PROGRAM MAIN
VAR
	tpImAPLC : TP;
END_VAR

////////////////////////////////////////////////////////////
// Logger test code
tpImAPLC();
IF NOT tpImAPLC.Q THEN
	fbLogMessage(i_sMsg:='Hello world, I am a PLC', i_eSevr:=Info, i_eSubsystem:=E_Subsystem.VACUUM);
	tpImAPLC(IN:= FALSE ); tpImAPLC(IN:= TRUE);
END_IF

END_PROGRAM

(* stored: Version 1.1.0.1, ProductVersion 3.1.4018.5
   POU MAIN: Id {d4dea680-4b5c-47cf-a536-e57c3bc8ef76}, SpecialFunc None *)
